// TIA Portal V20 export
TYPE "typeCmHmiInterfaceSoftCam"
// stored: Access Published, Namespace Unit1.Em2
   STRUCT
      jrOutPnPLeftAxisX : "Unit1.Em2.typeCmHmiInterfaceSoftCamjrOutPnPLeftAxisX";
      jrOutPnPLeftAxisZ : "Unit1.Em2.typeCmHmiInterfaceSoftCamjrOutPnPLeftAxisZ";
      jrOutPnPRightAxisX : "Unit1.Em2.typeCmHmiInterfaceSoftCamjrOutPnPRightAxisX";
      jrOutPnPRightAxisZ : "Unit1.Em2.typeCmHmiInterfaceSoftCamjrOutPnPRightAxisZ";
   END_STRUCT;
END_TYPE
